PROGRAM PRG_READ_List
VAR
	fbUA_ConnectEx			: UA_Connect;
	SessionConnectInfoEx	: ST_UASessionConnectInfo;
	sOpcUA_URL				: STRING(MAX_STRING_LENGTH);
	nConnectionHdl			: DWORD;

	fbUA_GetNamespaceIndex 	: UA_GetNamespaceIndex;
	nNamespaceIndex			: UINT;
	fbUA_NodeGetHandleList	: UA_NodeGetHandleList;
	
	NodeIDs					: ARRAY [1..nMaxNodeIDsInList] OF ST_UANodeID;
	nNodeHdls				: ARRAY [1..nMaxNodeIDsInList] OF DWORD;

	fbUA_ReadList			: UA_ReadList;
	NodeIDCount				: UINT := 2;
	NodeHdlCount			: UINT := 2; 
	stIndexRange			: ARRAY [1..nMaxIndexRange] OF ST_UAIndexRange;
	nIndexRangeCount		: UINT;
	stNodeAddInfo			: ARRAY [1..nMaxNodeIDsInList] OF ST_UANodeAdditionalInfo;
	stReadListData			: ST_ReadListData; // memory block must contain the Data[], NodeErrorIDs[], TimeStamps[] and cbData_R[]
	cbData					: ARRAY [1..nMaxNodeIDsInList] OF UDINT; (* Bytes to be actually Read *)
	cbData_R				: UDINT;
	cbDataTotal				: UDINT; 
	
	fbUA_NodeReleaseHandleList	: UA_NodeReleaseHandleList;

	fbUA_Disconnect		: UA_Disconnect;

	iState		: INT;
	bTest		: BOOL:= TRUE;
	bDone		: BOOL;
	bBusy		: BOOL;
	bError		: BOOL;
	nErrorID	: DWORD;
END_VAR


CASE iState OF
0:	(* idle *)
	IF bTest THEN
		bTest		:= FALSE;
		bError		:= FALSE;
		nErrorID	:= 0;

		SessionConnectInfoEx.tConnectTimeout 		:= T#1M;
		SessionConnectInfoEx.tSessionTimeout 		:= T#1M;
		SessionConnectInfoEx.sApplicationName		:= '';
		SessionConnectInfoEx.eSecurityMode 			:= eUASecurityMsgMode_None;
		SessionConnectInfoEx.eSecurityPolicyUri 	:= eUASecurityPolicy_None;
		SessionConnectInfoEx.eTransportProfileUri 	:= eUATransportProfileUri_UATcp;

		iState	:= iState + 1;
	END_IF

1:	(* open UA session *)
	fbUA_ConnectEx(
		Execute				:= TRUE,
		ServerURL			:= sOpcUaServerUrl,
		SessionConnectInfo  := SessionConnectInfoEx,
		Timeout				:= T#2M,
		ConnectionHdl		=> nConnectionHdl
	);

	IF NOT fbUA_ConnectEx.Busy THEN
		fbUA_ConnectEx(Execute := FALSE);

		IF NOT fbUA_ConnectEx.Error THEN
			(* session open *)
			iState := iState + 1;
		ELSE
			bError			:= TRUE;
			nErrorID		:= fbUA_ConnectEx.ErrorID;
			nConnectionHdl	:= 0;
			iState 			:= 0; (* idle *)
		END_IF
	END_IF


2:	(* GetNS Index *)
	fbUA_GetNamespaceIndex(
		Execute			:= TRUE,
		ConnectionHdl	:= nConnectionHdl,
		NamespaceUri	:= sNamespaceUri,
		NamespaceIndex	=> nNamespaceIndex
	);

	IF NOT fbUA_GetNamespaceIndex.Busy THEN
		fbUA_GetNamespaceIndex(Execute := FALSE);
		IF NOT fbUA_GetNamespaceIndex.Error THEN
			(* session closed *)
			iState 		:= iState + 1; (* idle *)
		ELSE
			bError		:= TRUE;
			nErrorID	:= fbUA_GetNamespaceIndex.ErrorID;
			iState 		:= 6; (* idle *)
		END_IF
	END_IF


3:	(* Get Node Handle *)
	
	NodeIDs[1].eIdentifierType := eUAIdentifierType_String;
	NodeIDs[1].nNamespaceIndex := nNamespaceIndex;
	NodeIDs[1].sIdentifier	:= 'MAIN.iVar1';
	
	NodeIDs[2].eIdentifierType := eUAIdentifierType_String;
	NodeIDs[2].nNamespaceIndex := nNamespaceIndex;
	NodeIDs[2].sIdentifier	:= 'MAIN.iVar2';

	fbUA_NodeGetHandleList(
		Execute			:= TRUE,
		ConnectionHdl	:= nConnectionHdl,
		NodeIDCount 	:= NodeIDCount,
		NodeIDs			:= NodeIDs,
		NodeHdls		=> nNodeHdls
	);

	IF NOT fbUA_NodeGetHandleList.Busy THEN
		fbUA_NodeGetHandleList(Execute := FALSE);

		IF NOT fbUA_NodeGetHandleList.Error THEN
			(* session closed *)
			iState 		:= iState + 1; (* idle *)
		ELSE
			bError		:= TRUE;
			nErrorID	:= fbUA_NodeGetHandleList.ErrorID;
			iState 		:= 6; (* idle *)
		END_IF
	END_IF

	
4: 	(* UA_Read *)
	cbData[1] := SIZEOF(stReadListData.nIntVar1);
	cbData[2] := SIZEOF(stReadListData.nIntVar2);
	cbDataTotal := SIZEOF(stReadListData);
	fbUA_ReadList(
		Execute			:= TRUE,
		ConnectionHdl	:= nConnectionHdl,
		NodeHdlCount	:= NodeHdlCount, // 2
		NodeHdls		:= nNodeHdls,
		stNodeAddInfo 	:= stNodeAddInfo,
		pVariable		:= ADR(stReadListData),
		cbData			:= cbData ,
		cbDataTotal		:= cbDataTotal		
		);

	IF NOT fbUA_ReadList.Busy THEN
		fbUA_ReadList( Execute := FALSE, cbData_R => cbData_R);

		IF NOT fbUA_ReadList.Error THEN
			(* session closed *)
			iState 		:= iState + 1; (* idle *)
		ELSE
			bError		:= TRUE;
			nErrorID	:= fbUA_ReadList.ErrorID;
			iState 		:= 6; (* idle *)
		END_IF
	END_IF


5:	(* Release Node Handle *)
	fbUA_NodeReleaseHandleList(
		Execute			:= TRUE,
		ConnectionHdl	:= nConnectionHdl,
		NodeHdlCount	:= NodeHdlCount,
		NodeHdls		:= nNodeHdls
	);

	IF NOT fbUA_NodeReleaseHandleList.Busy THEN
		fbUA_NodeReleaseHandleList(Execute := FALSE);

		IF NOT fbUA_NodeReleaseHandleList.Error THEN
			(* session closed *)
			iState 		:= iState + 1; (* idle *)
		ELSE
			bError		:= TRUE;
			nErrorID	:= fbUA_NodeReleaseHandleList.ErrorID;
			iState 		:= 6; (* idle *)
		END_IF
	END_IF


6:	(* close session *)
	fbUA_Disconnect(
		Execute			:= TRUE,
		ConnectionHdl	:= nConnectionHdl
	);

	IF NOT fbUA_Disconnect.Busy THEN
		fbUA_Disconnect(Execute := FALSE);
		bBusy := FALSE;
		IF NOT fbUA_Disconnect.Error THEN
			(* session closed *)
			iState 		:= 0; (* idle *)
			IF NOT bError THEN 
				bDone 	:= TRUE;
			END_IF
		ELSE
			bError			:= TRUE;
			nErrorID		:= fbUA_Disconnect.ErrorID;
			iState 			:= 0; (* idle *)
			nConnectionHdl	:= 0;
		END_IF
	END_IF
END_CASE

END_PROGRAM

(* stored: Version 1.1.0.1, ProductVersion 3.1.4024.3
   POU PRG_READ_List: Id {bd420e17-ea8f-4bb9-8bb3-35ac6d1cefa6}, SpecialFunc None *)
